INTERFACE I_RunObjects

METHOD Abort : BOOL
VAR_INPUT
END_VAR
VAR	
	i: INT;
END_VAR
END_METHOD

METHOD PUBLIC  Cycle : HRESULT
VAR_INPUT
END_VAR
VAR	
	i: INT;
END_VAR
END_METHOD

METHOD Initialise : HRESULT
VAR
	i : INT;
END_VAR
END_METHOD

METHOD Initialise_Ordered : HRESULT
VAR
	i : INT;
END_VAR
END_METHOD

METHOD Reset : HRESULT
VAR_INPUT
END_VAR
VAR	
	i: INT;
END_VAR
END_METHOD

END_INTERFACE

(* stored: Version 1.1.0.1
   Itf I_RunObjects: Id {61a2c5d3-0237-411f-8fd6-63b56ee659b9}
   Method Abort: Id {68d1c22b-b062-4ba5-af4e-be1c5aac2012}
   Method Cycle: Id {d3354a45-fc19-4351-8bac-e55f3d6a6b07}
   Method Initialise: Id {de761ae2-8c67-469f-9061-c94caa53bd35}
   Method Initialise_Ordered: Id {3fecbf72-28eb-4bcc-8029-8c43c7eea37a}
   Method Reset: Id {63e64e98-d635-4279-a162-64cc55a71604} *)
